(* IEC 61131-3 sources: AXOpen/src/components.cognex.vision/ctrl/src/AxoInsight/v_24_0_0 (part 2) *)

            //*************Soft event*****************
            SoftEventTask.IsDisabled :=  RestoreTask.IsBusy() OR ClearInspectionResultsTask.IsBusy() OR TriggerTask.IsBusy() OR ChangeJobByNameTask.IsBusy() OR ChangeJobByNumberTask.IsBusy() OR SendUserDataTask.IsBusy();
            IF SoftEventTask.StartTriggered() THEN
                Status.Action.Id :=  UINT#150;
            END_IF;
            Messenger.ActivateOnCondition(ULINT#150,SoftEventTask.IsBusy(), eAxoMessageCategory#Info);
            Messenger.ActivateOnCondition(ULINT#151,SoftEventTask.IsDone(), eAxoMessageCategory#Info);
            IF SoftEventTask.Execute(THIS) THEN
                IF _progress = 0 THEN
                    Status.Error.Id := UINT#0;
                    TaskMessenger.Restore();
                    THIS.CallTimers(FALSE);
                    _progress := 350;
                END_IF;

                IF _progress = 350 THEN
                    THIS.CallTimers(FALSE);
                    IF _softEventNumber > UINT#7 THEN
                        TaskMessenger.Activate( UINT#550, eAxoMessageCategory#Warning);
                        Status.Error.Id :=      UINT#550;
                        SoftEventTask.ThrowWhen(TRUE);
                    ELSE
                        _progress := 351;
                    END_IF;
                END_IF;

                IF _progress = 351 THEN
                    IF _infoTimer.output THEN
                        TaskMessenger.Activate( UINT#551, eAxoMessageCategory#Warning);
                        Status.Error.Id :=      UINT#551;
                    END_IF;
                    _progress := 352;
                END_IF;

                IF _progress = 352 THEN
                    IF _infoTimer.output THEN
                        TaskMessenger.Activate( UINT#552, eAxoMessageCategory#Warning);
                        Status.Error.Id :=      UINT#552;
                    END_IF;

                    SoftEventControl.TriggerSoftEvent.Data[_softEventNumber] := TRUE;
                    SoftEventControl.TriggerSoftEvent.ToggleDataChangedFlag();
                    IF SoftEventStatus.TriggerSoftEventAcknowledge.Data[_softEventNumber] THEN
                        SoftEventStatus.TriggerSoftEventAcknowledge.ToggleDataChangedFlag();
                        THIS.CallTimers(FALSE);
                        _progress := 353;
                    END_IF;
                END_IF;

                IF _progress = 353 THEN
                    IF _infoTimer.output THEN
                        TaskMessenger.Activate( UINT#553, eAxoMessageCategory#Warning);
                        Status.Error.Id :=      UINT#553;
                    END_IF;

                    SoftEventControl.TriggerSoftEvent.Data[_softEventNumber] := FALSE;
                    SoftEventControl.TriggerSoftEvent.ToggleDataChangedFlag();
                    IF NOT SoftEventStatus.TriggerSoftEventAcknowledge.Data[_softEventNumber] THEN
                        SoftEventStatus.TriggerSoftEventAcknowledge.ToggleDataChangedFlag();
                        THIS.CallTimers(FALSE);
                        _progress := 354;
                    END_IF;
                END_IF;

                IF _progress = 354 THEN
                    SoftEventTask.DoneWhen(TRUE);
                    _progress := 0;
                END_IF;

                THIS.CallTimers(TRUE);
                SoftEventTask.ThrowWhen(_errorTimer.output);
                Status.Action.Id := TO_UINT(_progress);
            END_IF;
            IF SoftEventTask.DoneReached() THEN
                Status.Action.Id :=  UINT#151;
                Status.Error.Id :=  UINT#0;
            ELSIF SoftEventTask.ErrorOccured() THEN
                Status.Action.Id :=  UINT#10050;
                Status.Error.Id  :=  UINT#10050;
            ELSIF SoftEventTask.AbortTriggered() THEN
                Status.Action.Id :=  UINT#10051;
                Status.Error.Id  :=  UINT#10051;
            END_IF;
            Messenger.ActivateOnCondition(ULINT#10050,SoftEventTask.HasError(), eAxoMessageCategory#Error);
            Messenger.ActivateOnCondition(ULINT#10051,SoftEventTask.IsAborted(), eAxoMessageCategory#Error);
            Messenger.ActivateOnCondition(ULINT#152,SoftEventTask.RestoreTriggered() , eAxoMessageCategory#Error);
            IF SoftEventTask.RestoreTriggered() AND _progress >= 350 AND _progress <= 359 THEN
                Status.Action.Id :=  UINT#152;
                _progress := 0;
            END_IF;
            //******************************************

            //*************SendUserData*****************
            SendUserDataTask.IsDisabled :=   RestoreTask.IsBusy() OR ClearInspectionResultsTask.IsBusy() OR TriggerTask.IsBusy() OR ChangeJobByNameTask.IsBusy() OR ChangeJobByNumberTask.IsBusy()  OR SoftEventTask.IsBusy();
            IF SendUserDataTask.StartTriggered() THEN
                Status.Action.Id :=  UINT#160;
            END_IF;
            Messenger.ActivateOnCondition(ULINT#160,SendUserDataTask.IsBusy(), eAxoMessageCategory#Info);
            Messenger.ActivateOnCondition(ULINT#161,SendUserDataTask.IsDone(), eAxoMessageCategory#Info);
            IF SendUserDataTask.Execute(THIS) THEN
                IF _progress = 0 THEN
                    Status.Error.Id := UINT#0;
                    TaskMessenger.Restore();
                    THIS.CallTimers(FALSE);
                    _progress := 360;
                END_IF;

                IF _progress = 360 THEN
                    IF _infoTimer.output THEN
                        TaskMessenger.Activate( UINT#560, eAxoMessageCategory#Warning);
                        Status.Error.Id :=      UINT#560;
                    END_IF;
                    IF THIS.SetUserDataAsString(UserDataToSent,UserDataOffset) THEN
                        THIS.CallTimers(FALSE);
                        _progress := 361;
                    END_IF;
                END_IF;

                IF _progress = 361 THEN
                    SendUserDataTask.DoneWhen(TRUE);
                    _progress := 0;
                END_IF;

                THIS.CallTimers(TRUE);
                SendUserDataTask.ThrowWhen(_errorTimer.output);
                Status.Action.Id := TO_UINT(_progress);
            END_IF;
            IF SendUserDataTask.DoneReached() THEN
                Status.Action.Id :=  UINT#161;
                Status.Error.Id :=  UINT#0;
            ELSIF SendUserDataTask.ErrorOccured() THEN
                Status.Action.Id :=  UINT#10060;
                Status.Error.Id  :=  UINT#10060;
            ELSIF SoftEventTask.AbortTriggered() THEN
                Status.Action.Id :=  UINT#10061;
                Status.Error.Id  :=  UINT#10061;
            END_IF;
            Messenger.ActivateOnCondition(ULINT#10060,SendUserDataTask.HasError(), eAxoMessageCategory#Error);
            Messenger.ActivateOnCondition(ULINT#10061,SendUserDataTask.IsAborted(), eAxoMessageCategory#Error);
            Messenger.ActivateOnCondition(ULINT#162,SendUserDataTask.RestoreTriggered() , eAxoMessageCategory#Error);
            IF SendUserDataTask.RestoreTriggered() AND _progress >= 360 AND _progress <= 369 THEN
                Status.Action.Id :=  UINT#162;
                _progress := 0;
            END_IF;
            //******************************************

            //***********Update outputs ****************
            _data_1[0].%X0              :=      AcquisitionControl.TriggerEnable;
            _data_1[0].%X1              :=      AcquisitionControl.Trigger;
            _data_1[0].%X2              :=      AcquisitionControl.ClearExposureComplete;
            _data_1[0].%X7              :=      AcquisitionControl.SetOffline;

            _retVal := Siemens.Simatic.S71500.DistributedIO.WriteData(_hwIdAcquisitionControl,_data_1);
            IF _retVal > WORD#0 THEN
                Messenger.Activate(UINT#1231, eAxoMessageCategory#ProgrammingError);
                Status.Error.Id := UINT#1231;
                RETURN;
            END_IF;

            _data_1[0].%X0               :=      InspectionControl.EnableResultsBuffering;
            _data_1[0].%X1               :=      InspectionControl.AcknowledgeInspectionResults;
            _data_1[0].%X2               :=      InspectionControl.ExtendedUserDataSet;
            _data_1[0].%X3               :=      InspectionControl.ExecuteCommand;
            _data_1[0].%X7               :=      InspectionControl.ClearError;

            _retVal := Siemens.Simatic.S71500.DistributedIO.WriteData(_hwIdInspectionControl,_data_1);
            IF _retVal > WORD#0 THEN
                Messenger.Activate(UINT#1232, eAxoMessageCategory#ProgrammingError);
                Status.Error.Id := UINT#1232;
                RETURN;
            END_IF;

            _data_2[0]                    :=      CommandControl.Command.%B1;
            _data_2[1]                    :=      CommandControl.Command.%B0;

            _retVal := Siemens.Simatic.S71500.DistributedIO.WriteData(_hwIdCommandControl,_data_2);
            IF _retVal > WORD#0 THEN
                Messenger.Activate(UINT#1233, eAxoMessageCategory#ProgrammingError);
                Status.Error.Id := UINT#1233;
                RETURN;
            END_IF;

            _data_1[0].%X0                  :=      SoftEventControl.TriggerSoftEvent.Data[0];
            _data_1[0].%X1                  :=      SoftEventControl.TriggerSoftEvent.Data[1];
            _data_1[0].%X2                  :=      SoftEventControl.TriggerSoftEvent.Data[2];
            _data_1[0].%X3                  :=      SoftEventControl.TriggerSoftEvent.Data[3];
            _data_1[0].%X4                  :=      SoftEventControl.TriggerSoftEvent.Data[4];
            _data_1[0].%X5                  :=      SoftEventControl.TriggerSoftEvent.Data[5];
            _data_1[0].%X6                  :=      SoftEventControl.TriggerSoftEvent.Data[6];
            _data_1[0].%X7                  :=      SoftEventControl.TriggerSoftEvent.Data[7];

            _retVal := Siemens.Simatic.S71500.DistributedIO.WriteData(_hwIdSoftEventControl,_data_1);
            IF _retVal > WORD#0 THEN
                Messenger.Activate(UINT#1234, eAxoMessageCategory#ProgrammingError);
                Status.Error.Id := UINT#1234;
                RETURN;
            END_IF;

            IF _hwIdUserDataSlot_7 <> WORD#0 THEN
                _invalidDataSize := NOT (   _UserDataSize_Slot_7 = UINT#16  OR
                                            _UserDataSize_Slot_7 = UINT#32  OR
                                            _UserDataSize_Slot_7 = UINT#64  OR
                                            _UserDataSize_Slot_7 = UINT#128 OR
                                            _UserDataSize_Slot_7 = UINT#254 );
                IF _invalidDataSize THEN
                    Messenger.Activate(UINT#1235, eAxoMessageCategory#ProgrammingError);
                    Status.Error.Id := UINT#1235;
                    RETURN;
                END_IF;
                IF (UserData.DataChanged <> _UserDataChanged) THEN
                    IF _UserDataSize_Slot_7 = UINT#16 THEN
                        FOR _index := 0 TO 15 DO
                            _data_16[_index] := UserData.Data[_index];
                        END_FOR;
                        _retVal := Siemens.Simatic.S71500.DistributedIO.WriteData(_hwIdUserDataSlot_7 ,_data_16);
                        IF _retVal > WORD#0 THEN
                            Messenger.Activate(UINT#1236, eAxoMessageCategory#ProgrammingError);
                            Status.Error.Id := UINT#1236;
                            RETURN;
                        END_IF;
                    ELSIF _UserDataSize_Slot_7 = UINT#32 THEN
                        FOR _index := 0 TO 31 DO
                            _data_32[_index] := UserData.Data[_index];
                        END_FOR;
                        _retVal := Siemens.Simatic.S71500.DistributedIO.WriteData(_hwIdUserDataSlot_7 ,_data_32);
                        IF _retVal > WORD#0 THEN
                            Messenger.Activate(UINT#1237, eAxoMessageCategory#ProgrammingError);
                            Status.Error.Id := UINT#1237;
                            RETURN;
                        END_IF;
                    ELSIF _UserDataSize_Slot_7 = UINT#64 THEN
                        FOR _index := 0 TO 63 DO
                            _data_64[_index] := UserData.Data[_index];
                        END_FOR;
                        _retVal := Siemens.Simatic.S71500.DistributedIO.WriteData(_hwIdUserDataSlot_7 ,_data_64);
                        IF _retVal > WORD#0 THEN
                            Messenger.Activate(UINT#1238, eAxoMessageCategory#ProgrammingError);
                            Status.Error.Id := UINT#1238;
                            RETURN;
                        END_IF;
                    ELSIF _UserDataSize_Slot_7 = UINT#128 THEN
                        FOR _index := 0 TO 127 DO
                            _data_128[_index] := UserData.Data[_index];
                        END_FOR;
                        _retVal := Siemens.Simatic.S71500.DistributedIO.WriteData(_hwIdUserDataSlot_7 ,_data_128);
                        IF _retVal > WORD#0 THEN
                            Messenger.Activate(UINT#1239, eAxoMessageCategory#ProgrammingError);
                            Status.Error.Id := UINT#1239;
                            RETURN;
                        END_IF;
                    ELSIF _UserDataSize_Slot_7 = UINT#254 THEN
                        FOR _index := 0 TO 253 DO
                            _data_254[_index] := UserData.Data[_index];
                        END_FOR;
                        _retVal := Siemens.Simatic.S71500.DistributedIO.WriteData(_hwIdUserDataSlot_7 ,_data_254);
                        IF _retVal > WORD#0 THEN
                            Messenger.Activate(UINT#1240, eAxoMessageCategory#ProgrammingError);
                            Status.Error.Id := UINT#1240;
                            RETURN;
                        END_IF;
                    END_IF;
                END_IF;
            END_IF;

            IF _hwIdUserDataSlot_8 <> WORD#0 THEN
                _invalidDataSize := NOT (   _UserDataSize_Slot_8 = UINT#16  OR
                                            _UserDataSize_Slot_8 = UINT#32  OR
                                            _UserDataSize_Slot_8 = UINT#64  OR
                                            _UserDataSize_Slot_8 = UINT#128 OR
                                            _UserDataSize_Slot_8 = UINT#254 );
                IF _invalidDataSize THEN
                    Messenger.Activate(UINT#1241, eAxoMessageCategory#ProgrammingError);
                    Status.Error.Id := UINT#1241;
                    RETURN;
                END_IF;
                IF (UserData.DataChanged <> _UserDataChanged) THEN
                    _offset := TO_INT(_UserDataSize_Slot_7);
                    IF _UserDataSize_Slot_8 = UINT#16 THEN
                        FOR _index := 0 TO 15 DO
                            _data_16[_index] := UserData.Data[_index+_offset];
                        END_FOR;
                        _retVal := Siemens.Simatic.S71500.DistributedIO.WriteData(_hwIdUserDataSlot_8 ,_data_16);
                        IF _retVal > WORD#0 THEN
                            Messenger.Activate(UINT#1242, eAxoMessageCategory#ProgrammingError);
                            Status.Error.Id := UINT#1242;
                            RETURN;
                        END_IF;
                    ELSIF _UserDataSize_Slot_8 = UINT#32 THEN
                        FOR _index := 0 TO 31 DO
                            _data_32[_index] := UserData.Data[_index+_offset];
                        END_FOR;
                        _retVal := Siemens.Simatic.S71500.DistributedIO.WriteData(_hwIdUserDataSlot_8 ,_data_32);
                        IF _retVal > WORD#0 THEN
                            Messenger.Activate(UINT#1243, eAxoMessageCategory#ProgrammingError);
                            Status.Error.Id := UINT#1243;
                            RETURN;
                        END_IF;
                    ELSIF _UserDataSize_Slot_8 = UINT#64 THEN
                        FOR _index := 0 TO 63 DO
                            _data_64[_index] := UserData.Data[_index+_offset];
                        END_FOR;
                        _retVal := Siemens.Simatic.S71500.DistributedIO.WriteData(_hwIdUserDataSlot_8 ,_data_64);
                        IF _retVal > WORD#0 THEN
                            Messenger.Activate(UINT#1244, eAxoMessageCategory#ProgrammingError);
                            Status.Error.Id := UINT#1244;
                            RETURN;
                        END_IF;
                    ELSIF _UserDataSize_Slot_8 = UINT#128 THEN
                        FOR _index := 0 TO 127 DO
                            _data_128[_index] := UserData.Data[_index+_offset];
                        END_FOR;
                        _retVal := Siemens.Simatic.S71500.DistributedIO.WriteData(_hwIdUserDataSlot_8 ,_data_128);
                        IF _retVal > WORD#0 THEN
                            Messenger.Activate(UINT#1245, eAxoMessageCategory#ProgrammingError);
                            Status.Error.Id := UINT#1245;
                            RETURN;
                        END_IF;
                    ELSIF _UserDataSize_Slot_8 = UINT#254 THEN
                        FOR _index := 0 TO 253 DO
                            _data_254[_index] := UserData.Data[_index+_offset];
                        END_FOR;
                        _retVal := Siemens.Simatic.S71500.DistributedIO.WriteData(_hwIdUserDataSlot_8 ,_data_254);
                        IF _retVal > WORD#0 THEN
                            Messenger.Activate(UINT#1246, eAxoMessageCategory#ProgrammingError);
                            Status.Error.Id := UINT#1246;
                            RETURN;
                        END_IF;
                    END_IF;
                END_IF;
            END_IF;

            IF _hwIdUserDataSlot_9 <> WORD#0 THEN
                _invalidDataSize := NOT (   _UserDataSize_Slot_9 = UINT#16  OR
                                            _UserDataSize_Slot_9 = UINT#32  OR
                                            _UserDataSize_Slot_9 = UINT#64  OR
                                            _UserDataSize_Slot_9 = UINT#128 OR
                                            _UserDataSize_Slot_9 = UINT#254 );
                IF _invalidDataSize THEN
                    Messenger.Activate(UINT#1247, eAxoMessageCategory#ProgrammingError);
                    Status.Error.Id := UINT#1247;
                    RETURN;
                END_IF;
                IF (UserData.DataChanged <> _UserDataChanged) THEN
                    _offset := TO_INT(_UserDataSize_Slot_7)+TO_INT(_UserDataSize_Slot_8);
                    IF _UserDataSize_Slot_9 = UINT#16 THEN
                        FOR _index := 0 TO 15 DO
                            _data_16[_index] := UserData.Data[_index+_offset];
                        END_FOR;
                        _retVal := Siemens.Simatic.S71500.DistributedIO.WriteData(_hwIdUserDataSlot_9 ,_data_16);
                        IF _retVal > WORD#0 THEN
                            Messenger.Activate(UINT#1248, eAxoMessageCategory#ProgrammingError);
                            Status.Error.Id := UINT#1248;
                            RETURN;
                        END_IF;
                    ELSIF _UserDataSize_Slot_9 = UINT#32 THEN
                        FOR _index := 0 TO 31 DO
                            _data_32[_index] := UserData.Data[_index+_offset];
                        END_FOR;
                        _retVal := Siemens.Simatic.S71500.DistributedIO.WriteData(_hwIdUserDataSlot_9 ,_data_32);
                        IF _retVal > WORD#0 THEN
                            Messenger.Activate(UINT#1249, eAxoMessageCategory#ProgrammingError);
                            Status.Error.Id := UINT#1249;
                            RETURN;
                        END_IF;
                    ELSIF _UserDataSize_Slot_9 = UINT#64 THEN
                        FOR _index := 0 TO 63 DO
                            _data_64[_index] := UserData.Data[_index+_offset];
                        END_FOR;
                        _retVal := Siemens.Simatic.S71500.DistributedIO.WriteData(_hwIdUserDataSlot_9 ,_data_64);
                        IF _retVal > WORD#0 THEN
                            Messenger.Activate(UINT#1250, eAxoMessageCategory#ProgrammingError);
                            Status.Error.Id := UINT#1250;
                            RETURN;
                        END_IF;
                    ELSIF _UserDataSize_Slot_9 = UINT#128 THEN
                        FOR _index := 0 TO 127 DO
                            _data_128[_index] := UserData.Data[_index+_offset];
                        END_FOR;
                        _retVal := Siemens.Simatic.S71500.DistributedIO.WriteData(_hwIdUserDataSlot_9 ,_data_128);
                        IF _retVal > WORD#0 THEN
                            Messenger.Activate(UINT#1251, eAxoMessageCategory#ProgrammingError);
                            Status.Error.Id := UINT#1251;
                            RETURN;
                        END_IF;
                    ELSIF _UserDataSize_Slot_9 = UINT#254 THEN
                        FOR _index := 0 TO 253 DO
                            _data_254[_index] := UserData.Data[_index+_offset];
                        END_FOR;
                        _retVal := Siemens.Simatic.S71500.DistributedIO.WriteData(_hwIdUserDataSlot_9 ,_data_254);
                        IF _retVal > WORD#0 THEN
                            Messenger.Activate(UINT#1252, eAxoMessageCategory#ProgrammingError);
                            Status.Error.Id := UINT#1252;
                            RETURN;
                        END_IF;
                    END_IF;
                END_IF;
            END_IF;

            IF _hwIdUserDataSlot_10 <> WORD#0 THEN
                _invalidDataSize := NOT (   _UserDataSize_Slot_10 = UINT#16  OR
                                            _UserDataSize_Slot_10 = UINT#32  OR
                                            _UserDataSize_Slot_10 = UINT#64  OR
                                            _UserDataSize_Slot_10 = UINT#128 OR
                                            _UserDataSize_Slot_10 = UINT#254 );
                IF _invalidDataSize THEN
                    Messenger.Activate(UINT#1253, eAxoMessageCategory#ProgrammingError);
                    Status.Error.Id := UINT#1253;
                    RETURN;
                END_IF;
                IF (UserData.DataChanged <> _UserDataChanged) THEN
                    _offset := TO_INT(_UserDataSize_Slot_7)+TO_INT(_UserDataSize_Slot_8)+TO_INT(_UserDataSize_Slot_9);
                    IF _UserDataSize_Slot_10 = UINT#16 THEN
                        FOR _index := 0 TO 15 DO
                            _data_16[_index] := UserData.Data[_index+_offset];
                        END_FOR;
                        _retVal := Siemens.Simatic.S71500.DistributedIO.WriteData(_hwIdUserDataSlot_10 ,_data_16);
                        IF _retVal > WORD#0 THEN
                            Messenger.Activate(UINT#1254, eAxoMessageCategory#ProgrammingError);
                            Status.Error.Id := UINT#1254;
                            RETURN;
                        END_IF;
                    ELSIF _UserDataSize_Slot_10 = UINT#32 THEN
                        FOR _index := 0 TO 31 DO
                            _data_32[_index] := UserData.Data[_index+_offset];
                        END_FOR;
                        _retVal := Siemens.Simatic.S71500.DistributedIO.WriteData(_hwIdUserDataSlot_10 ,_data_32);
                        IF _retVal > WORD#0 THEN
                            Messenger.Activate(UINT#1255, eAxoMessageCategory#ProgrammingError);
                            Status.Error.Id := UINT#1255;
                            RETURN;
                        END_IF;
                    ELSIF _UserDataSize_Slot_10 = UINT#64 THEN
                        FOR _index := 0 TO 63 DO
                            _data_64[_index] := UserData.Data[_index+_offset];
                        END_FOR;
                        _retVal := Siemens.Simatic.S71500.DistributedIO.WriteData(_hwIdUserDataSlot_10 ,_data_64);
                        IF _retVal > WORD#0 THEN
                            Messenger.Activate(UINT#1256, eAxoMessageCategory#ProgrammingError);
                            Status.Error.Id := UINT#1256;
                            RETURN;
                        END_IF;
                    ELSIF _UserDataSize_Slot_10 = UINT#128 THEN
                        FOR _index := 0 TO 127 DO
                            _data_128[_index] := UserData.Data[_index+_offset];
                        END_FOR;
                        _retVal := Siemens.Simatic.S71500.DistributedIO.WriteData(_hwIdUserDataSlot_10 ,_data_128);
                        IF _retVal > WORD#0 THEN
                            Messenger.Activate(UINT#1257, eAxoMessageCategory#ProgrammingError);
                            Status.Error.Id := UINT#1257;
                            RETURN;
                        END_IF;
                    ELSIF _UserDataSize_Slot_10 = UINT#254 THEN
                        FOR _index := 0 TO 253 DO
                            _data_254[_index] := UserData.Data[_index+_offset];
                        END_FOR;
                        _retVal := Siemens.Simatic.S71500.DistributedIO.WriteData(_hwIdUserDataSlot_10 ,_data_254);
                        IF _retVal > WORD#0 THEN
                            Messenger.Activate(UINT#1258, eAxoMessageCategory#ProgrammingError);
                            Status.Error.Id := UINT#1258;
                            RETURN;
                        END_IF;
                    END_IF;
                END_IF;
            END_IF;

            _UserDataChanged := UserData.DataChanged;  //TODO check the functionality in case of multiple user data slots
            Config.UserDataSize := _UserDataSize;
        END_METHOD

        ///<summary>
		/// Clears the inspection results.
        ///</summary>
        METHOD PUBLIC ClearInspectionResults : IAxoTaskState
            ClearInspectionResults := ClearInspectionResultsTask.Invoke(THIS);;
        END_METHOD

        ///<summary>
		/// Triggers the reading sequence and waits for results.
        ///</summary>
        METHOD PUBLIC Trigger : IAxoTaskState
            Trigger := TriggerTask.Invoke(THIS);
        END_METHOD

        ///<summary>
		/// Changes the sensor job using job number.
        ///</summary>
        METHOD PUBLIC ChangeJob : IAxoTaskState
            VAR_INPUT
                Job : UINT;
            END_VAR
            _jobNumber := Job;
            ChangeJob := ChangeJobByNumberTask.Invoke(THIS);
        END_METHOD

        ///<summary>
		/// Changes the sensor job using job name.
        ///</summary>
        METHOD PUBLIC ChangeJob : IAxoTaskState
            VAR_INPUT
                Job : STRING;
            END_VAR
            _jobName := Job;
            ChangeJob := ChangeJobByNameTask.Invoke(THIS);
        END_METHOD

        ///<summary>
		/// Triggers the soft event.
        ///</summary>
        METHOD PUBLIC SoftEvent : IAxoTaskState
            VAR_INPUT
                EventNumber : UINT;
            END_VAR
            _softEventNumber := EventNumber;
            SoftEvent := SoftEventTask.Invoke(THIS);
        END_METHOD

        METHOD PRIVATE CallTimers
            VAR_INPUT
                signal : BOOL;
            END_VAR

            _infoTimer.OnDelay(THIS, signal , Config.InfoTime);
            _errorTimer.OnDelay(THIS, signal , Config.ErrorTime );
        END_METHOD

        METHOD INTERNAL AppendSuffix :STRING
            VAR_INPUT
                jobName : STRING;
            END_VAR
            VAR
                position : INT;
            END_VAR
            position := LengthOf(jobName) - 4;
            IF EndOf(jobName, 4) <> '.job' THEN
                AppendSuffix := Concat(jobName,'.job');
            ELSE
                AppendSuffix := jobName;
            END_IF;
        END_METHOD

        METHOD INTERNAL SetUserDataAsString :   BOOL
            VAR_INPUT
                inValue     :   STRING;
                inPosition  :   UINT;
            END_VAR
            VAR
                _index : UINT;
                _size : UINT;
                _maxIndex : UINT;
                _data : ARRAY[0..255] OF BYTE;
            END_VAR

            SetUserDataAsString := FALSE;

            _size := TO_UINT(LengthOf(inValue));

            _maxIndex := UINT#255;

            IF (inPosition +_size) >= Config.UserDataSize THEN
                Messenger.Activate(UINT#716, eAxoMessageCategory#Error);
                Status.Error.Id := UINT#716;
                RETURN;
            END_IF;

            IF (inPosition +_size) > _maxIndex THEN
                Messenger.Activate(UINT#717, eAxoMessageCategory#Error);
                Status.Error.Id := UINT#717;
                RETURN;
            END_IF;

            Serialize(UINT#0, inValue, _data);
            FOR	_index := UINT#0 TO _size BY UINT#1 DO
                UserData.Data[(inPosition + _index)] := _data[_index + UINT#1];
            END_FOR;

            FOR	_index := inPosition +_size TO _maxIndex BY UINT#1 DO
                UserData.Data[_index] := BYTE#0;
            END_FOR;
            UserData.ToggleDataChangedFlag();

            SetUserDataAsString := TRUE;
        END_METHOD

        ///<summary>
		/// Custom logic for the manual control.
        ///</summary>
        METHOD PROTECTED OVERRIDE ManualControl
            _jobName := RequiredJobName;
            _jobNumber := RequiredJobNumber;
            _softEventNumber := RequiredSoftEventNumber;
        END_METHOD

        ///<summary>
		/// Restores this instance .
        ///</summary>
        METHOD PUBLIC OVERRIDE Restore
            VAR
                _index : INT;
            END_VAR
            _progress := 0;
            Status.Action.Id := UINT#0;
            Status.Error.Id  := UINT#0;
            Status.CurrentJobName := '';
            Messenger.Restore();
            TaskMessenger.Restore();

            ClearInspectionResultsTask.Restore();
            TriggerTask.Restore();
            ChangeJobByNameTask.Restore();
            ChangeJobByNumberTask.Restore();
            SoftEventTask.Restore();
            SendUserDataTask.Restore();
            HardwareDiagnosticsTask.Restore();

            UserDataToSent := '';
            UserDataOffset := UINT#0;

            RequiredJobName := '';
            RequiredJobNumber := UINT#0;

            Results.InspectionID                            :=  UINT#0;
            Results.ResultCode                              :=  UINT#0;

            FOR _index := 0 TO 249 DO
                InspectionResults.Data[_index] := BYTE#0;
            END_FOR;
            InspectionResults.ToggleDataChangedFlag();

            AcquisitionControl.TriggerEnable                :=  FALSE;
            AcquisitionControl.Trigger					    :=  FALSE;
            AcquisitionControl.ClearExposureComplete        :=  AcquisitionStatus.ExposureComplete;
            AcquisitionControl.SetOffline                   :=  FALSE;

            InspectionControl.EnableResultsBuffering        :=  FALSE;
            InspectionControl.AcknowledgeInspectionResults  :=  FALSE;
            InspectionControl.ExtendedUserDataSet           :=  FALSE;
            InspectionControl.ExecuteCommand                :=  FALSE;
            InspectionControl.ClearError                    :=  InspectionStatus.Error;

            CommandControl.Command                          :=  UINT#0;

            SoftEventControl.TriggerSoftEvent.Data[0]       :=  FALSE;
            SoftEventControl.TriggerSoftEvent.Data[1]       :=  FALSE;
            SoftEventControl.TriggerSoftEvent.Data[2]       :=  FALSE;
            SoftEventControl.TriggerSoftEvent.Data[3]       :=  FALSE;
            SoftEventControl.TriggerSoftEvent.Data[4]       :=  FALSE;
            SoftEventControl.TriggerSoftEvent.Data[5]       :=  FALSE;
            SoftEventControl.TriggerSoftEvent.Data[6]       :=  FALSE;
            SoftEventControl.TriggerSoftEvent.Data[7]       :=  FALSE;

            FOR _index := 0 TO 253 DO
                UserData.Data[_index] := BYTE#0;
            END_FOR;
            UserData.ToggleDataChangedFlag();

            IF NOT AcquisitionStatus.ExposureComplete AND NOT InspectionStatus.Error THEN
                Status.Action.Id := UINT#50;
                RestoreTask.DoneWhen(TRUE);
            END_IF;
        END_METHOD

    END_CLASS
END_NAMESPACE
